FUNCTION_BLOCK FB_CreateDir_V2
VAR_INPUT
	InPath 				: T_Maxstring;
	InExe				: BOOL;
END_VAR
VAR_OUTPUT
	OutExiste			: BOOL;
	OutCompleted		: BOOL;
	OutError			: BOOL;
	OutErrorId			: UDINT;
	OutBusy				: BOOL;
END_VAR
VAR
	CreateDir			: FB_CreateDir;	
	
	Trig_Start			: RS;
	Trig				: R_TRIG;
	
	
END_VAR

Trig(CLK := InExe);
//OutCompleted := NOT Trig.Q AND NOT CreateDir.bBusy AND NOT CreateDir.bError;
Trig_Start(SET := Trig.Q);

CreateDir(
	sNetId := '', 
	sPathName := InPath,
	bExecute := Trig.Q
	);
	
IF Trig_Start.Q1 AND NOT CreateDir.bBusy AND (CreateDir.nErrId = 16#723 OR CreateDir.nErrId = 16#70C ) THEN
	createDir(bExecute := FALSE);
	OutExiste := TRUE;
	OutCompleted := TRUE;
	Trig(CLK := FALSE);
	Trig_Start( RESET1 := OutCompleted OR OutError);
	Trig_Start( RESET1 := FALSE);
ELSIF NOT Trig.Q AND Trig_Start.Q1 AND NOT CreateDir.bBusy AND NOT CreateDir.bError THEN
	OutCompleted := TRUE;
	CreateDir(bExecute := FALSE);
	Trig(CLK := FALSE);
	Trig_Start( RESET1 := OutCompleted OR OutError);
	Trig_Start( RESET1 := FALSE);
ELSIF CreateDir.bError THEN
	OutError := TRUE;
	OutErrorId := CreateDir.nErrid;
	CreateDir(bExecute := FALSE);
	Trig(CLK := FALSE);
	Trig_Start( RESET1 := OutCompleted OR OutError);
	Trig_Start( RESET1 := FALSE);

END_IF

OutBusy := Trig_Start.Q1;

END_FUNCTION_BLOCK

(* stored: Version 1.1.0.1, ProductVersion 3.1.4024.6
   POU FB_CreateDir_V2: Id {2b1a4923-505e-4c69-8a46-4d9c5bb7f307}, SpecialFunc None *)
